TYPE ST_Test3 :
STRUCT
	sString: STRING(10) := '';
	fReal: REAL;
	iInt: INT;
	nByte: BYTE;
	bCheckbox: BOOL;
	arrBool: ARRAY[1..5] OF BOOL;
END_STRUCT
END_TYPE

(* stored: Version 1.1.0.1, ProductVersion 3.1.0.36
   DUT ST_Test3: Id {d05d384e-edc0-425e-878c-0effe91f299c} *)
